% RSLogix 500 project TASK4.RSS, saved by version 8.30.00.16 %
PROJECT "UNTITLED"    % processor: Bul.1763 MicroLogix 1100 Series B %

PROGRAM FILES
  LAD 2   6 rungs

DATA FILES
  O0 OUTPUT  4 elements
  I1 INPUT  6 elements
  S2 STATUS  66 elements
  B3 BINARY  1 elements
  T4 TIMER  1 elements
  C5 COUNTER  1 elements
  R6 CONTROL  1 elements
  N7 INTEGER  1 elements
  F8 FLOAT  1 elements

LADDER 2
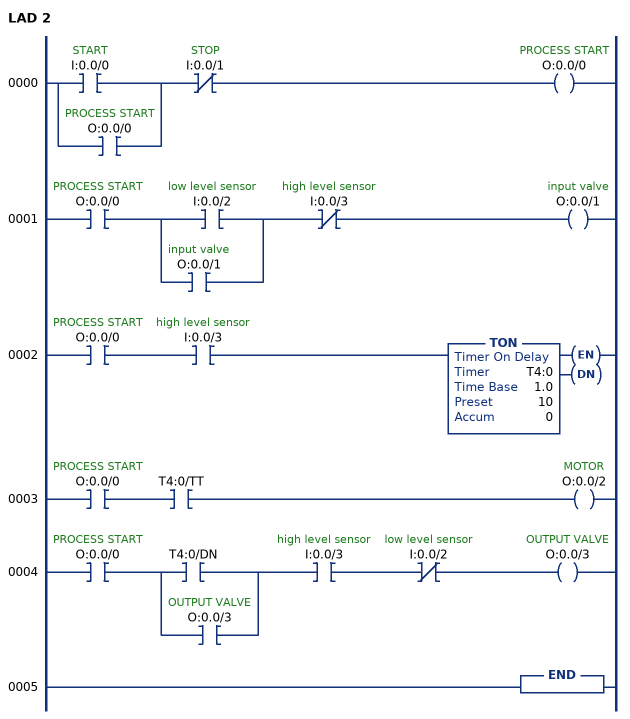
% Rung: 0 %
SOR BST XIC I:0.0/0 NXB XIC O:0.0/0 BND XIO I:0.0/1 OTE O:0.0/0 EOR
%   I:0.0/0  "START" %
%   O:0.0/0  "PROCESS START" %
%   I:0.0/1  "STOP" %
% Rung: 1 %
SOR XIC O:0.0/0 BST XIC I:0.0/2 NXB XIC O:0.0/1 BND XIO I:0.0/3 OTE O:0.0/1 EOR
%   O:0.0/0  "PROCESS START" %
%   I:0.0/2  "low level sensor" %
%   O:0.0/1  "input valve" %
%   I:0.0/3  "high level sensor" %
% Rung: 2 %
SOR XIC O:0.0/0 XIC I:0.0/3 TON T4:0 1.0 10 0 EOR
%   O:0.0/0  "PROCESS START" %
%   I:0.0/3  "high level sensor" %
% Rung: 3 %
SOR XIC O:0.0/0 XIC T4:0/TT OTE O:0.0/2 EOR
%   O:0.0/0  "PROCESS START" %
%   O:0.0/2  "MOTOR" %
% Rung: 4 %
SOR XIC O:0.0/0 BST XIC T4:0/DN NXB XIC O:0.0/3 BND XIC I:0.0/3 XIO I:0.0/2 OTE O:0.0/3 EOR
%   O:0.0/0  "PROCESS START" %
%   O:0.0/3  "OUTPUT VALVE" %
%   I:0.0/3  "high level sensor" %
%   I:0.0/2  "low level sensor" %
% Rung: 5 %
SOR END EOR

DATA TABLE (non-zero values as saved)
DATA T4
% .PRE .ACC %
% T4:0 % 10 0
